// TwinCAT 3 PLC project Untitled1
// ProgramVersion: 3.1.4024.0
// libraries:
//   Tc2_Standard, * (Beckhoff Automation GmbH)
//   Tc2_System, * (Beckhoff Automation GmbH)
//   Tc3_Module, * (Beckhoff Automation GmbH)
// project tree:
//   / Gestionnaire de visualisation.TcVMO (not stored), GlobalTextList.TcGTLO, PlcTask.TcTTO
//   GVLs/ GVL.TcGVL
//   POUs/ MAIN.TcPOU
//   VISUs/ Visualization.TcVIS
// real-time tasks:
//   TASK PlcTask: cycle T#10ms, priority 20, ADS port 350
// I/O:
//   DEVICE Périphérique 1 (EtherCAT), AmsNetId 192.168.1.191.2.1
//     Terme 1 (EK1100) [EK1100 EtherCAT Coupler (2A E-Bus)]
//       Terme 2 (EL2008) [EL2008 8Ch. Dig. Output 24V, 0.5A]
//       Terme 3 (EL1008) [EL1008 8Ch. Dig. Input 24V, 3ms]
//       Terme 4 (EL3255) [EL3255 5Ch. potentiometer measurement with sensor supply]
//       Terme 5 (EL9011) [EL9011 End Terminal]

CONFIGURATION Untitled1
    RESOURCE PLC ON TwinCAT3
        TASK PlcTask(INTERVAL := T#10ms, PRIORITY := 20);
        PROGRAM MAIN WITH PlcTask : MAIN;
    END_RESOURCE
END_CONFIGURATION

// ---- GVLs/GVL.TcGVL
{attribute 'qualified_only'}
VAR_GLOBAL

    BoutonVirtuel : BOOL := FALSE;
    Lumiere : BOOL := FALSE;
	iPushCounter : UINT := 0 ;
	
END_VAR

// ---- POUs/MAIN.TcPOU
PROGRAM MAIN
VAR
    rTrig : R_TRIG;
END_VAR


// Détection front montant
rTrig(CLK := GVL.BoutonVirtuel);

IF GVL.BoutonVirtuel THEN
    GVL.Lumiere := TRUE;
ELSE
    GVL.Lumiere := FALSE;
END_IF;

// Incrément seulement sur appui
IF rTrig.Q THEN
    GVL.iPushCounter := GVL.iPushCounter + 1;
END_IF;

END_PROGRAM

// ---- VISUs/Visualization.TcVIS
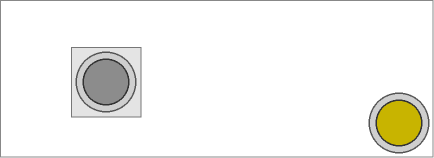
VISUALIZATION Visualization  // 434x158
    PushSwitch (71,47 70x70), variable: GVL.BoutonVirtuel, behaviour: TOGGLE, style: Switch-PushSwitch-Gray
    Lamp1 (364,88 70x70), variable: GVL.Lumiere, style: Lamp-Lamp1-Yellow
END_VISUALIZATION
